RoboDK station: Sidestringers.rdk

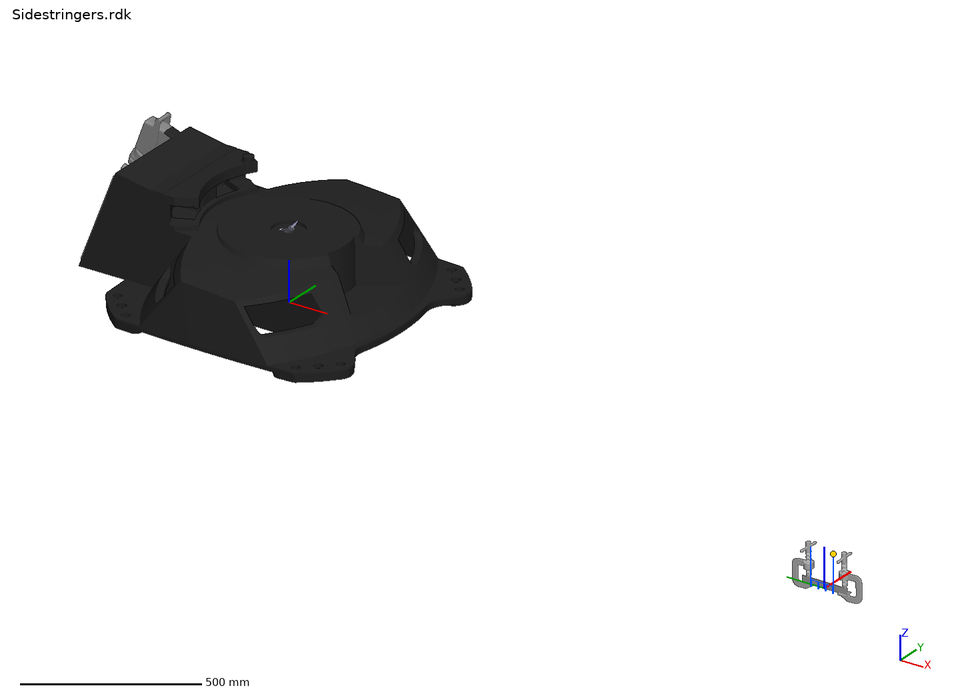
[picture v0: the station drawn from its stored meshes, robots at their saved joint values, targets as dots, program paths as lines]
Station Sidestringers (saved by RoboDK 5.2.3). Poses are relative to the parent item; angles as X-Y-Z fixed-axis rotations.
  - frame KUKA KR 210 R2700 extra Base at (0, 0, 0) mm
    - robot KUKA KR 210 R2700 extra: 6 axes, payload 210 kg, reach 2696 mm, repeatability 0.06 mm, weight 1068 kg
        joint limits [-185, -140, -120, -350, -125, -350] to [185, -5, 155, 350, 125, 350]; home [0, -90, 90, 0, 0, 0]; saved at [-0.458, -33.509, 109.285, 179.312, 24.776, -179.731]
      - tool Spindle, TCP at (32, 0, 260) mm, rotated rx 0 ry 39 rz 0 deg, size 157.3 x 72 x 259.9 mm
  - frame Frame 2 at (1800, 0, -372.68) mm, rotated rx 0 ry 0 rz 90 deg
    - object sidestringer at (0, 0, 0) mm, rotated rx 0 ry 0 rz -90 deg, size 152 x 20 x 20 mm, geometry from sidestringer.stl
    - object sidestringers at (0, 0, 0) mm, rotated rx 0 ry 0 rz 180 deg, 4 curves, geometry from Point 4
  - machining project Point settings: rotZ(0) | rotX(0)*rotY(0) | rotz(0) | onStart | onPathStart | onApproach | onPoint | onRetract | onFinish | SetRPM(%1) | SetTool(%1) | Extruder(%1) | default | default | OutOnMov(%1) | OutOffMov(%1) | onPathFinish | M_RunCode(%1) | riverData=C:\Windows\System32\Driv | PS_BROWSER_APP_PROFILE_STRING=Inter | PS_BROWSER_USER_PROFILE_STRING=Defa | OCALAPPDATA=C:\Users\jbert\AppData\Loc | OneDrive=C:\Users\jbert\O | Path=C:\Program Files (x86)\NVIDIA Corpora
  - program Point (31 instructions, listed below)
  - object FinalClamp at (1857.38, 12.44, -311.02) mm, rotated rx 153.25 ry 89.01 rz 67.76 deg, size 145.3 x 71.1 x 72 mm, geometry from FinalClamp.stp
  - object FinalClamp2 at (1737.84, 11.11, -311.03) mm, rotated rx -87.7 ry 89.16 rz 3.46 deg, size 145.3 x 71.1 x 72 mm, geometry from FinalClamp.stp
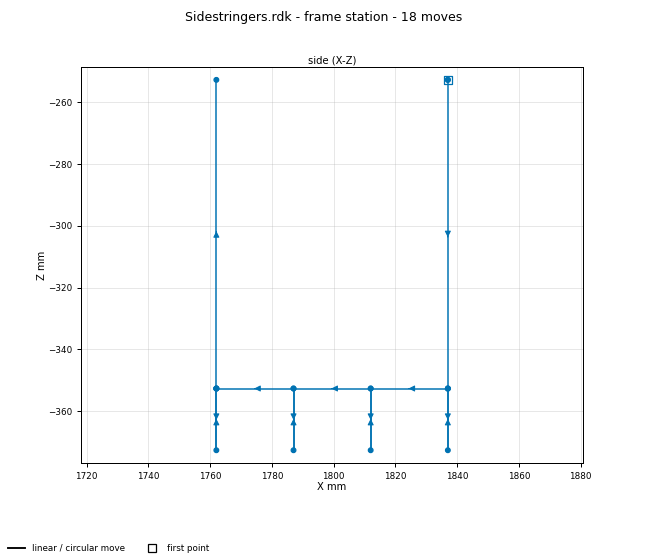
[picture p0: tool path of Sidestringers.rdk in frame station, 18 of 18 moves have a stored position in this frame; points joined in program order, loops and branches not executed]

--- program Point (robot KUKA KR 210 R2700 extra) ---
  Smooth(1)
  Set speed (1000.0 mm/s)
  Set Ref.: Frame 2
  Set Tool: Spindle
  Show Spindle
  MoveJ 1 to (-12.5, -37, 120) mm, rotated rx -180 ry 0 rz -90 deg; joints [-0.481, -34.261, 113.27, 179.355, 28.009, -179.805]
  MoveL 2 to (-12.5, -37, 120) mm, rotated rx -180 ry 0 rz -90 deg; joints [-0.481, -34.261, 113.27, 179.355, 28.009, -179.805]
  MoveL 3 to (-12.5, -37, 20) mm, rotated rx 180 ry 0 rz -90 deg; joints [-0.481, -28.858, 110.599, 179.408, 30.741, -179.865]
  MoveL 4 to (-12.5, -37, 20) mm, rotated rx 180 ry 0 rz -90 deg; joints [-0.481, -28.858, 110.599, 179.408, 30.741, -179.865]
  Set speed (50.0 mm/s)
  MoveL 5 to (-12.5, -37, 0) mm, rotated rx 180 ry 0 rz -90 deg; joints [-0.481, -27.788, 110.018, 179.416, 31.23, -179.875]
  MoveL 6 to (-12.5, -37, 20) mm, rotated rx 180 ry 0 rz -90 deg; joints [-0.481, -28.858, 110.599, 179.408, 30.741, -179.865]
  Set speed (1000.0 mm/s)
  MoveL 7 to (-12.5, -12, 20) mm, rotated rx 180 ry 0 rz -90 deg; joints [-0.473, -28.698, 109.312, 179.398, 29.614, -179.844]
  Set speed (50.0 mm/s)
  MoveL 8 to (-12.5, -12, 0) mm, rotated rx 180 ry 0 rz -90 deg; joints [-0.473, -27.639, 108.735, 179.406, 30.097, -179.854]
  MoveL 9 to (-12.5, -12, 20) mm, rotated rx 180 ry 0 rz -90 deg; joints [-0.473, -28.698, 109.312, 179.398, 29.614, -179.844]
  Set speed (1000.0 mm/s)
  MoveL 10 to (-12.5, 13, 20) mm, rotated rx 180 ry 0 rz -90 deg; joints [-0.465, -28.513, 108.008, 179.386, 28.495, -179.822]
  Set speed (50.0 mm/s)
  MoveL 11 to (-12.5, 13, 0) mm, rotated rx -180 ry 0 rz -90 deg; joints [-0.465, -27.466, 107.436, 179.395, 28.971, -179.833]
  MoveL 12 to (-12.5, 13, 20) mm, rotated rx 180 ry 0 rz -90 deg; joints [-0.465, -28.513, 108.008, 179.386, 28.495, -179.822]
  Set speed (1000.0 mm/s)
  MoveL 13 to (-12.5, 38, 20) mm, rotated rx -180 ry 0 rz -90 deg; joints [-0.458, -28.304, 106.687, 179.373, 27.383, -179.8]
  Set speed (50.0 mm/s)
  MoveL 14 to (-12.5, 38, 0) mm, rotated rx -180 ry 0 rz -90 deg; joints [-0.458, -27.268, 106.12, 179.383, 27.852, -179.81]
  MoveL 15 to (-12.5, 38, 20) mm, rotated rx -180 ry 0 rz -90 deg; joints [-0.458, -28.304, 106.687, 179.373, 27.383, -179.8]
  MoveL 16 to (-12.5, 38, 20) mm, rotated rx -180 ry 0 rz -90 deg; joints [-0.458, -28.304, 106.687, 179.373, 27.383, -179.8]
  Set speed (1000.0 mm/s)
  MoveL 17 to (-12.5, 38, 20) mm, rotated rx -180 ry 0 rz -90 deg; joints [-0.458, -28.304, 106.687, 179.373, 27.383, -179.8]
  MoveL 18 to (-12.5, 38, 120) mm, rotated rx 180 ry 0 rz -90 deg; joints [-0.458, -33.509, 109.285, 179.312, 24.776, -179.731]
